(* PLC project paper-machine, Generated TextualNotationConverter 1.0 *)
(* stored: creationDateTime 2025-07-30T12:00:00, modificationDateTime 2025-01-30T12:00:00 *)

FUNCTION_BLOCK ANALOG_IN
  VAR_INPUT
    Name : STRING;
    Description : STRING;
    Raw_Signal : REAL;
    PV_High : REAL;
    PV_Low : REAL;
    Scaling_Slope : REAL;
    Scaling_Offset : REAL;
    Alarm_Enable : BOOL;
  END_VAR
  VAR_OUTPUT
    PV : REAL;
    High_Alarm : BOOL;
    Low_Alarm : BOOL;
    General_Fault : BOOL;
  END_VAR

            
          
END_FUNCTION_BLOCK

FUNCTION_BLOCK BOOL_IN
  VAR_INPUT
    Name : STRING;
    Description : STRING;
    Bool_In : BOOL;
    Alarm_OnTrue : BOOL;
    Alarm_OnFalse : BOOL;
    Latch_Enable : BOOL;
    Reset_Latch : BOOL;
  END_VAR
  VAR_OUTPUT
    Bool_Out : BOOL;
    Alarm_Active : BOOL;
    Latched_Status : BOOL;
  END_VAR

            
          
END_FUNCTION_BLOCK

FUNCTION_BLOCK MOTOR_VSD
  VAR_INPUT
    Name : STRING;
    Description : STRING;
    Start_Cmd : BOOL;
    Stop_Cmd : BOOL;
    Speed_SP : REAL;
    Accel_Ramp : STRING;
    Decel_Ramp : STRING;
    Inhibit : BOOL;
  END_VAR
  VAR_OUTPUT
    Speed_Out : REAL;
    FB_Running : BOOL;
    FB_Fault : BOOL;
    FB_Ready : BOOL;
    FB_ActualSpeed : REAL;
    Alarm_Speed_Deviation : BOOL;
    Alarm_Comm_Fail : BOOL;
  END_VAR

            
          
END_FUNCTION_BLOCK

FUNCTION_BLOCK PID_BASIC
  VAR_INPUT
    Name : STRING;
    Description : STRING;
    AUTO : BOOL;
    PV : REAL;
    SP : REAL;
    MV_MIN : REAL;
    MV_MAX : REAL;
    X0 : REAL;
    KP : REAL;
    TR : REAL;
    TD : REAL;
    PV_High : REAL;
    PV_Low : REAL;
    Deviation_Limit : REAL;
    Inhibit : BOOL;
  END_VAR
  VAR_OUTPUT
    PV_High_Alarm : BOOL;
    PV_Low_Alarm : BOOL;
    Deviation_Alarm : BOOL;
    XOUT : REAL;
  END_VAR

            
          
END_FUNCTION_BLOCK

FUNCTION_BLOCK VALVE_ELECTRIC
  VAR_INPUT
    Name : STRING;
    Description : STRING;
    Control_Signal : REAL;
    Manual_Mode : BOOL;
    Manual_Position : REAL;
    Open_Limit : REAL;
    Close_Limit : REAL;
    Timeout : STRING;
    Inhibit : BOOL;
  END_VAR
  VAR_OUTPUT
    Valve_Position : REAL;
    Feedback_Pos : REAL;
    Valve_Moving : BOOL;
    Position_Error : BOOL;
    Alarm : BOOL;
  END_VAR

            
          
END_FUNCTION_BLOCK

FUNCTION_BLOCK VALVE_ON_OFF
  VAR_INPUT
    Name : STRING;
    Description : STRING;
    Open_Cmd : BOOL;
    Close_Cmd : BOOL;
    Timeout : STRING;
    Inhibit : BOOL;
  END_VAR
  VAR_OUTPUT
    FB_Opened : BOOL;
    FB_Closed : BOOL;
    Valve_Open_Out : BOOL;
    Valve_Close_Out : BOOL;
    Alarm_Position_Error : BOOL;
    Alarm_General : BOOL;
  END_VAR

            
          
END_FUNCTION_BLOCK

PROGRAM Section2
  VAR
    LT101_Flow_PV_m3ph : REAL;
    FC101_MV_Percent : REAL;
    HopperLevel_Above20 : BOOL;
  END_VAR
  VAR
    LT-101 : ANALOG_IN;
    FC-101 : PID_BASIC;
    M-102 : MOTOR_VSD;
    FV-106 : VALVE_ELECTRIC;
    XV-102 : VALVE_ON_OFF;
    XV-104 : VALVE_ON_OFF;
    XV-105 : VALVE_ON_OFF;
    ILK-FC-101-XV-102-OPEN : BOOL_IN;
    ILK-FC-101-XV-104-OPEN : BOOL_IN;
    ILK-FC-101-LT-101-VALID : BOOL_IN;
    PERM-M-102-LEVEL-ABOVE-20 : BOOL_IN;
    PERM-M-102-XV-105-CLOSED : BOOL_IN;
    M102RestartDelay_TON : TON;
  END_VAR
  VAR  (* added by the conversion: wires and edge detectors of the diagram *)
    _OR9_OUT : BOOL;
    _NOT10_OUT : BOOL;
    _AND3_OUT : BOOL;
  END_VAR

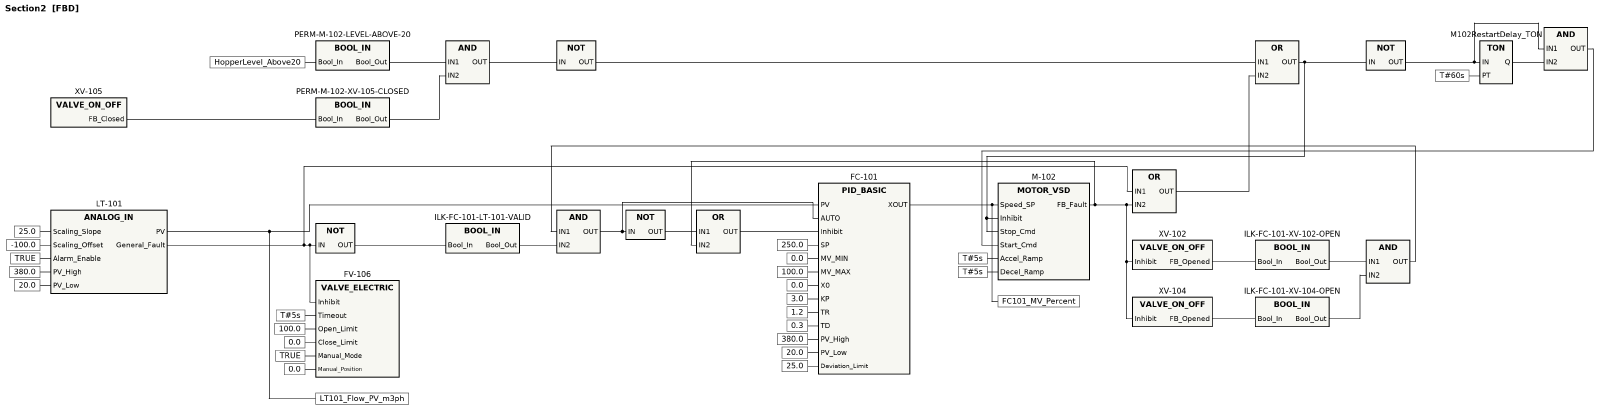
(* FBD diagram, written out as Structured Text *)
LT-101(Scaling_Slope := 25.0, Scaling_Offset := -100.0, Alarm_Enable := TRUE, PV_High := 380.0, PV_Low := 20.0);
PERM-M-102-LEVEL-ABOVE-20(Bool_In := HopperLevel_Above20);
XV-105();
PERM-M-102-XV-105-CLOSED(Bool_In := XV-105.FB_Closed);
_OR9_OUT := NOT (PERM-M-102-LEVEL-ABOVE-20.Bool_Out AND PERM-M-102-XV-105-CLOSED.Bool_Out) OR LT-101.General_Fault OR M-102.FB_Fault;
_NOT10_OUT := NOT _OR9_OUT;
M102RestartDelay_TON(IN := _NOT10_OUT, PT := T#60s);
M-102(Speed_SP := FC-101.XOUT, Inhibit := _OR9_OUT, Stop_Cmd := _OR9_OUT, Start_Cmd := _NOT10_OUT AND M102RestartDelay_TON.Q, Accel_Ramp := T#5s, Decel_Ramp := T#5s);
XV-102(Inhibit := M-102.FB_Fault);
ILK-FC-101-XV-102-OPEN(Bool_In := XV-102.FB_Opened);
XV-104(Inhibit := M-102.FB_Fault);
ILK-FC-101-XV-104-OPEN(Bool_In := XV-104.FB_Opened);
ILK-FC-101-LT-101-VALID(Bool_In := NOT LT-101.General_Fault);
_AND3_OUT := ILK-FC-101-XV-102-OPEN.Bool_Out AND ILK-FC-101-XV-104-OPEN.Bool_Out AND ILK-FC-101-LT-101-VALID.Bool_Out;
FC-101(PV := LT-101.PV, AUTO := _AND3_OUT, Inhibit := NOT _AND3_OUT OR M-102.FB_Fault, SP := 250.0, MV_MIN := 0.0, MV_MAX := 100.0, X0 := 0.0, KP := 3.0, TR := 1.2, TD := 0.3, PV_High := 380.0, PV_Low := 20.0, Deviation_Limit := 25.0);
FC101_MV_Percent := FC-101.XOUT;
LT101_Flow_PV_m3ph := LT-101.PV;
FV-106(Inhibit := LT-101.General_Fault, Timeout := T#5s, Open_Limit := 100.0, Close_Limit := 0.0, Manual_Mode := TRUE, Manual_Position := 0.0);
END_PROGRAM

FUNCTION_BLOCK DIGITAL_IN
  VAR_INPUT
    Name : STRING;
    Description : STRING;
    DI_Raw : BOOL;
    DebounceTime : STRING;
    EnableAlarm : BOOL;
  END_VAR
  VAR_OUTPUT
    DI_Out : BOOL;
    Fault_State : BOOL;
  END_VAR

            
          
END_FUNCTION_BLOCK

FUNCTION_BLOCK DUTY_STANDBY
  VAR_INPUT
    Name : STRING;
    Description : STRING;
    Enable : BOOL;
    StartRequest : BOOL;
    AlternateEnable : BOOL;
    ForcePumpA : BOOL;
    ForcePumpB : BOOL;
    DutyElapsed : BOOL;
    MinRunElapsed : BOOL;
    SwitchoverDelayElapsed : BOOL;
    StartTimeoutElapsed : BOOL;
    PumpA_RunFB : BOOL;
    PumpB_RunFB : BOOL;
    PumpA_Fault : BOOL;
    PumpB_Fault : BOOL;
    Reset : BOOL;
    Inhibit : BOOL;
  END_VAR
  VAR_OUTPUT
    CmdPumpA : BOOL;
    CmdPumpB : BOOL;
    ActiveIsA : BOOL;
    SwitchedDueToDuty : BOOL;
    SwitchedDueToFailure : BOOL;
    Alarm_FailedStart_A : BOOL;
    Alarm_FailedStart_B : BOOL;
    Alarm_NoAvailablePump : BOOL;
  END_VAR

            
          
END_FUNCTION_BLOCK

FUNCTION_BLOCK MOTOR_2SPD
  VAR_INPUT
    Name : STRING;
    Description : STRING;
    Start_Cmd : BOOL;
    Stop_Cmd : BOOL;
    Speed_High_Cmd : BOOL;
    Speed_Low_Cmd : BOOL;
    Inhibit : BOOL;
  END_VAR
  VAR_OUTPUT
    Motor_Start_Out : BOOL;
    FB_Running : BOOL;
    FB_Trip : BOOL;
    FB_HighSpeed : BOOL;
    FB_LowSpeed : BOOL;
    Alarm_Speed_Error : BOOL;
  END_VAR

            
          
END_FUNCTION_BLOCK

FUNCTION_BLOCK MOTOR_ON_OFF
  VAR_INPUT
    Name : STRING;
    Description : STRING;
    Start_Cmd : BOOL;
    Stop_Cmd : BOOL;
    Start_Delay : STRING;
    MinRunTime : STRING;
    Inhibit : BOOL;
  END_VAR
  VAR_OUTPUT
    Motor_Start_Out : BOOL;
    FB_Running : BOOL;
    FB_Trip : BOOL;
    Alarm_Start_Fail : BOOL;
    Alarm_Stop_Fail : BOOL;
  END_VAR

            
          
END_FUNCTION_BLOCK

FUNCTION_BLOCK RATIO_CONTROL
  VAR_INPUT
    Name : STRING;
    Description : STRING;
    Auto : BOOL;
    PrimaryPV : REAL;
    SecondaryPV : REAL;
    RatioSP : REAL;
    Bias : REAL;
    TrimKp : REAL;
    TrimTi : STRING;
    MV_MIN : REAL;
    MV_MAX : REAL;
    ManOut : REAL;
    Inhibit : BOOL;
  END_VAR
  VAR_OUTPUT
    SlaveSP : REAL;
    ActiveRatio : REAL;
    RatioErr : REAL;
  END_VAR

            
          
END_FUNCTION_BLOCK

FUNCTION_BLOCK SPLIT_RANGE
  VAR_INPUT
    Name : STRING;
    Description : STRING;
    IN : REAL;
    Split_Point : REAL;
    Output1_Start : REAL;
    Output1_End : REAL;
    Output2_Start : REAL;
    Output2_End : REAL;
  END_VAR
  VAR_OUTPUT
    OUT1 : REAL;
    OUT2 : REAL;
  END_VAR

            
          
END_FUNCTION_BLOCK

FUNCTION_BLOCK VOTING_ANALOG
  VAR_INPUT
    Name : STRING;
    Description : STRING;
    Input1 : REAL;
    Input2 : REAL;
    Input3 : REAL;
    Deviation_Limit : REAL;
    Voting_Scheme : STRING;
    EnableAlarm : BOOL;
    Inhibit : BOOL;
  END_VAR
  VAR_OUTPUT
    Voted_Output : REAL;
    Sensor1_Fault : BOOL;
    Sensor2_Fault : BOOL;
    Sensor3_Fault : BOOL;
    Alarm_Voting_Error : BOOL;
    Healthy_Sensors_Count : INT;
  END_VAR

            
          
END_FUNCTION_BLOCK

PROGRAM Section3
  VAR
    TIC104_RSP_to_FC203 : REAL;
    PIC101_RSP_to_FC202 : REAL;
    FC203_ControlSignal_SV203 : REAL;
    FC202_ControlSignal_FV202 : REAL;
  END_VAR
  VAR
    PT-101 : ANALOG_IN;
    TT-103 : ANALOG_IN;
    PIC-101 : PID_BASIC;
    TIC-104 : PID_BASIC;
    FC-202 : PID_BASIC;
    FC-203 : PID_BASIC;
    FV-202 : VALVE_ELECTRIC;
    SV-203 : VALVE_ELECTRIC;
  END_VAR
  VAR  (* added by the conversion: wires and edge detectors of the diagram *)
    _OR51_OUT : BOOL;
  END_VAR

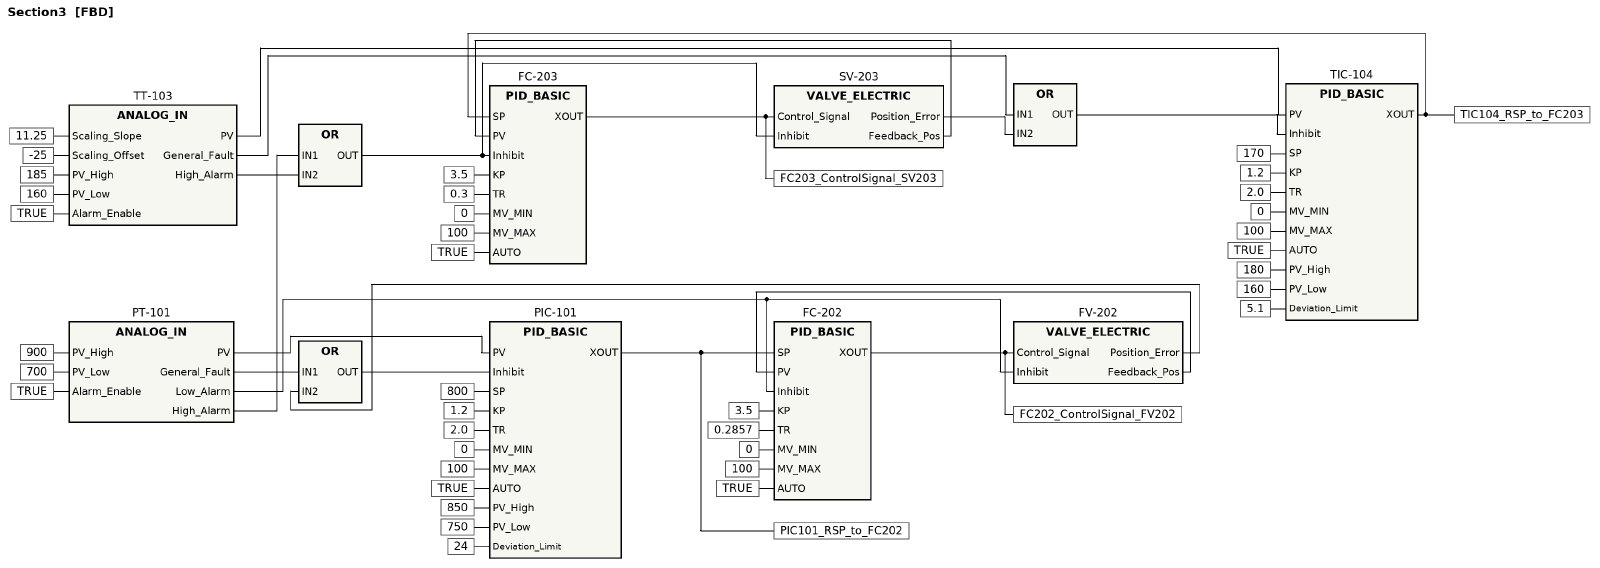
(* FBD diagram, written out as Structured Text *)
PT-101(PV_High := 900, PV_Low := 700, Alarm_Enable := TRUE);
FV-202(Control_Signal := FC-202.XOUT, Inhibit := PT-101.Low_Alarm);
PIC-101(PV := PT-101.PV, Inhibit := PT-101.General_Fault OR FV-202.Position_Error, SP := 800, KP := 1.2, TR := 2.0, MV_MIN := 0, MV_MAX := 100, AUTO := TRUE, PV_High := 850, PV_Low := 750, Deviation_Limit := 24);
FC-202(SP := PIC-101.XOUT, PV := FV-202.Feedback_Pos, Inhibit := PT-101.Low_Alarm, KP := 3.5, TR := 0.2857, MV_MIN := 0, MV_MAX := 100, AUTO := TRUE);
FC202_ControlSignal_FV202 := FC-202.XOUT;
TT-103(Scaling_Slope := 11.25, Scaling_Offset := -25, PV_High := 185, PV_Low := 160, Alarm_Enable := TRUE);
_OR51_OUT := PT-101.High_Alarm OR TT-103.High_Alarm;
SV-203(Control_Signal := FC-203.XOUT, Inhibit := _OR51_OUT);
TIC-104(PV := TT-103.PV, Inhibit := TT-103.General_Fault OR SV-203.Position_Error, SP := 170, KP := 1.2, TR := 2.0, MV_MIN := 0, MV_MAX := 100, AUTO := TRUE, PV_High := 180, PV_Low := 160, Deviation_Limit := 5.1);
FC-203(SP := TIC-104.XOUT, PV := SV-203.Feedback_Pos, Inhibit := _OR51_OUT, KP := 3.5, TR := 0.3, MV_MIN := 0, MV_MAX := 100, AUTO := TRUE);
FC203_ControlSignal_SV203 := FC-203.XOUT;
PIC101_RSP_to_FC202 := PIC-101.XOUT;
TIC104_RSP_to_FC203 := TIC-104.XOUT;
END_PROGRAM

PROGRAM Section4
  VAR
    PIT103_Pressure_PV : REAL;
    PT101_UpstreamPressure_PV : REAL;
    DT301_Density_PV : REAL;
    PIC104_MV_to_FV106 : REAL;
    FV106_Position_Feedback : REAL;
  END_VAR
  VAR
    PIT-103 : ANALOG_IN;
    PT-101 : ANALOG_IN;
    DT-301 : ANALOG_IN;
    PIC-104 : PID_BASIC;
    FV-106 : VALVE_ELECTRIC;
    XV-102 : VALVE_ON_OFF;
    XV-107 : VALVE_ON_OFF;
    XV-102-OPEN-LS : DIGITAL_IN;
    XV-107-OPEN-LS : DIGITAL_IN;
    ILK-FEED-PRESSURE-OK : BOOL_IN;
    ILK-OVERPRESSURE-TRIP : BOOL_IN;
    ILK-DENSITY-OK : BOOL_IN;
    ILK-XV102-OPEN : BOOL_IN;
    ILK-XV107-OPEN : BOOL_IN;
    ILK-SYSTEM-FAULT : BOOL_IN;
  END_VAR

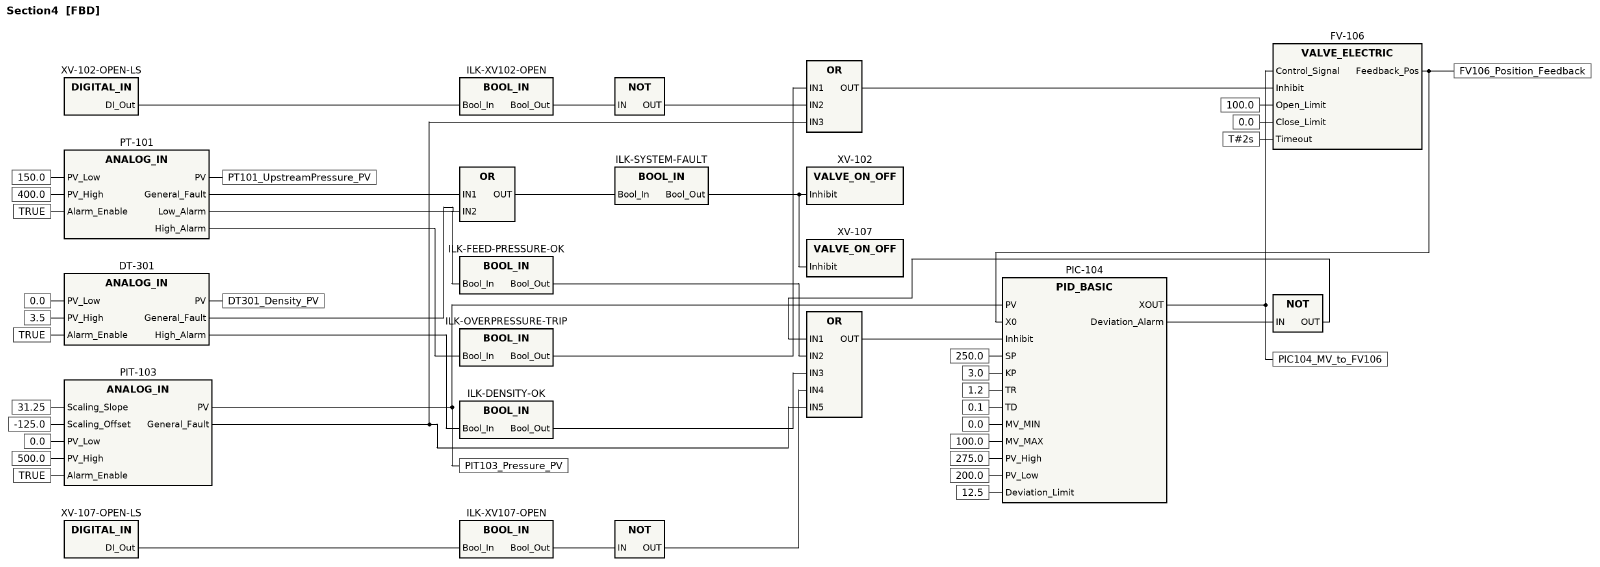
(* FBD diagram, written out as Structured Text *)
DT-301(PV_Low := 0.0, PV_High := 3.5, Alarm_Enable := TRUE);
DT301_Density_PV := DT-301.PV;
PIT-103(Scaling_Slope := 31.25, Scaling_Offset := -125.0, PV_Low := 0.0, PV_High := 500.0, Alarm_Enable := TRUE);
PT-101(PV_Low := 150.0, PV_High := 400.0, Alarm_Enable := TRUE);
ILK-FEED-PRESSURE-OK(Bool_In := PT-101.Low_Alarm);
ILK-DENSITY-OK(Bool_In := DT-301.High_Alarm);
XV-107-OPEN-LS();
ILK-XV107-OPEN(Bool_In := XV-107-OPEN-LS.DI_Out);
PIC-104(PV := PIT-103.PV, X0 := FV-106.Feedback_Pos, Inhibit := NOT PIC-104.Deviation_Alarm OR ILK-FEED-PRESSURE-OK.Bool_Out OR ILK-DENSITY-OK.Bool_Out OR NOT ILK-XV107-OPEN.Bool_Out OR PIT-103.General_Fault, SP := 250.0, KP := 3.0, TR := 1.2, TD := 0.1, MV_MIN := 0.0, MV_MAX := 100.0, PV_High := 275.0, PV_Low := 200.0, Deviation_Limit := 12.5);
ILK-OVERPRESSURE-TRIP(Bool_In := PT-101.High_Alarm);
XV-102-OPEN-LS();
ILK-XV102-OPEN(Bool_In := XV-102-OPEN-LS.DI_Out);
FV-106(Control_Signal := PIC-104.XOUT, Inhibit := ILK-OVERPRESSURE-TRIP.Bool_Out OR NOT ILK-XV102-OPEN.Bool_Out OR PIT-103.General_Fault, Open_Limit := 100.0, Close_Limit := 0.0, Timeout := T#2s);
FV106_Position_Feedback := FV-106.Feedback_Pos;
PIC104_MV_to_FV106 := PIC-104.XOUT;
PIT103_Pressure_PV := PIT-103.PV;
PT101_UpstreamPressure_PV := PT-101.PV;
ILK-SYSTEM-FAULT(Bool_In := PT-101.General_Fault OR DT-301.General_Fault);
XV-102(Inhibit := ILK-SYSTEM-FAULT.Bool_Out);
XV-107(Inhibit := ILK-SYSTEM-FAULT.Bool_Out);
END_PROGRAM

PROGRAM Section5
  VAR
    AT102_pH_PV : REAL;
    AT107_pH_PV : REAL;
    TIT106_Temperature_PV : REAL;
    FIT_UPSTREAM_Flow_PV : REAL;
    DPIT_FLOW_PV : REAL;
    PIT_DOWNSTREAM_Pressure_PV : REAL;
    LIT_TOWER_Level_PV : REAL;
    LIC102_MV_to_FV101 : REAL;
    TIC106_MV_to_FV103 : REAL;
    LIC104_Output_to_XV104 : REAL;
    FV101_Position_AO : REAL;
    FV103_Position_AO : REAL;
  END_VAR
  VAR
    AT-102 : ANALOG_IN;
    AT-107 : ANALOG_IN;
    TIT-106 : ANALOG_IN;
    FIT-UPSTREAM : ANALOG_IN;
    DPIT-FLOW : ANALOG_IN;
    PIT-DOWNSTREAM : ANALOG_IN;
    LIT-TOWER : ANALOG_IN;
    LIC-102 : PID_BASIC;
    TIC-106 : PID_BASIC;
    LIC-104 : PID_BASIC;
    FV-101 : VALVE_ELECTRIC;
    FV-103 : VALVE_ELECTRIC;
    XV-104 : VALVE_ON_OFF;
    INTERLOCK-FV101-UPSTREAM-FLOW-OK : BOOL_IN;
    INTERLOCK-LIC102-PH-SAFE : BOOL_IN;
    INTERLOCK-TIC106-TEMP-SAFE : BOOL_IN;
    INTERLOCK-LIC104-FLOW-OK : BOOL_IN;
    INTERLOCK-LIC104-PRESSURE-OK : BOOL_IN;
    PERMISSIVE-TOWER-LEVEL-OK : BOOL_IN;
  END_VAR

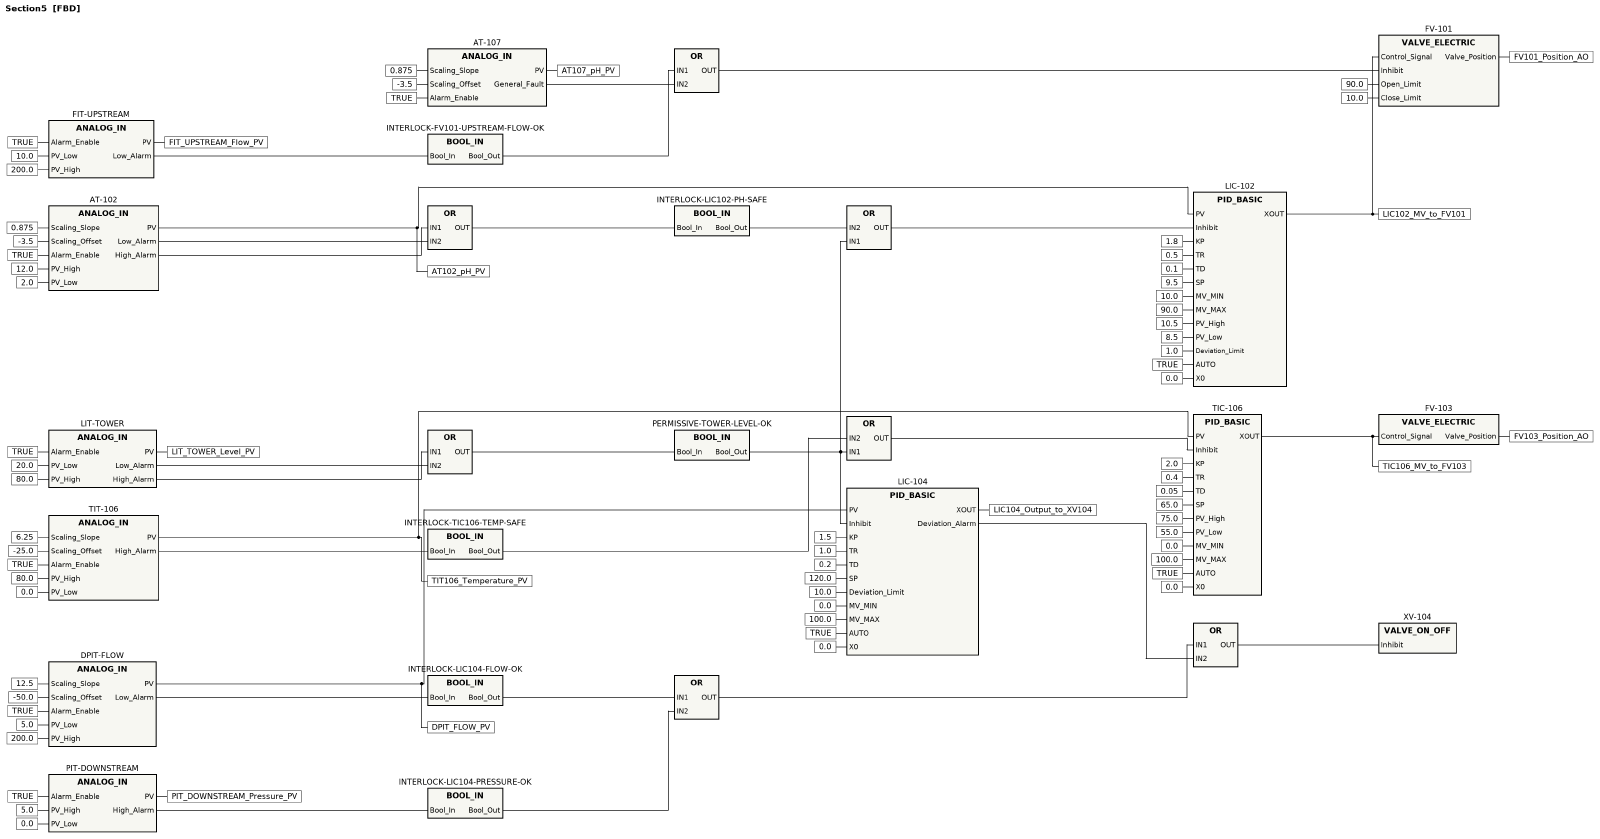
(* FBD diagram, written out as Structured Text *)
AT-102(Scaling_Slope := 0.875, Scaling_Offset := -3.5, Alarm_Enable := TRUE, PV_High := 12.0, PV_Low := 2.0);
AT102_pH_PV := AT-102.PV;
AT-107(Scaling_Slope := 0.875, Scaling_Offset := -3.5, Alarm_Enable := TRUE);
AT107_pH_PV := AT-107.PV;
DPIT-FLOW(Scaling_Slope := 12.5, Scaling_Offset := -50.0, Alarm_Enable := TRUE, PV_Low := 5.0, PV_High := 200.0);
DPIT_FLOW_PV := DPIT-FLOW.PV;
FIT-UPSTREAM(Alarm_Enable := TRUE, PV_Low := 10.0, PV_High := 200.0);
FIT_UPSTREAM_Flow_PV := FIT-UPSTREAM.PV;
INTERLOCK-LIC102-PH-SAFE(Bool_In := AT-102.High_Alarm OR AT-102.Low_Alarm);
LIT-TOWER(Alarm_Enable := TRUE, PV_Low := 20.0, PV_High := 80.0);
PERMISSIVE-TOWER-LEVEL-OK(Bool_In := LIT-TOWER.High_Alarm OR LIT-TOWER.Low_Alarm);
LIC-102(PV := AT-102.PV, Inhibit := INTERLOCK-LIC102-PH-SAFE.Bool_Out OR PERMISSIVE-TOWER-LEVEL-OK.Bool_Out, KP := 1.8, TR := 0.5, TD := 0.1, SP := 9.5, MV_MIN := 10.0, MV_MAX := 90.0, PV_High := 10.5, PV_Low := 8.5, Deviation_Limit := 1.0, AUTO := TRUE, X0 := 0.0);
INTERLOCK-FV101-UPSTREAM-FLOW-OK(Bool_In := FIT-UPSTREAM.Low_Alarm);
FV-101(Control_Signal := LIC-102.XOUT, Inhibit := INTERLOCK-FV101-UPSTREAM-FLOW-OK.Bool_Out OR AT-107.General_Fault, Open_Limit := 90.0, Close_Limit := 10.0);
FV101_Position_AO := FV-101.Valve_Position;
TIT-106(Scaling_Slope := 6.25, Scaling_Offset := -25.0, Alarm_Enable := TRUE, PV_High := 80.0, PV_Low := 0.0);
INTERLOCK-TIC106-TEMP-SAFE(Bool_In := TIT-106.High_Alarm);
TIC-106(PV := TIT-106.PV, Inhibit := INTERLOCK-TIC106-TEMP-SAFE.Bool_Out OR PERMISSIVE-TOWER-LEVEL-OK.Bool_Out, KP := 2.0, TR := 0.4, TD := 0.05, SP := 65.0, PV_High := 75.0, PV_Low := 55.0, MV_MIN := 0.0, MV_MAX := 100.0, AUTO := TRUE, X0 := 0.0);
FV-103(Control_Signal := TIC-106.XOUT);
FV103_Position_AO := FV-103.Valve_Position;
LIC102_MV_to_FV101 := LIC-102.XOUT;
LIC-104(PV := DPIT-FLOW.PV, Inhibit := PERMISSIVE-TOWER-LEVEL-OK.Bool_Out, KP := 1.5, TR := 1.0, TD := 0.2, SP := 120.0, Deviation_Limit := 10.0, MV_MIN := 0.0, MV_MAX := 100.0, AUTO := TRUE, X0 := 0.0);
LIC104_Output_to_XV104 := LIC-104.XOUT;
LIT_TOWER_Level_PV := LIT-TOWER.PV;
PIT-DOWNSTREAM(Alarm_Enable := TRUE, PV_High := 5.0, PV_Low := 0.0);
PIT_DOWNSTREAM_Pressure_PV := PIT-DOWNSTREAM.PV;
TIC106_MV_to_FV103 := TIC-106.XOUT;
TIT106_Temperature_PV := TIT-106.PV;
INTERLOCK-LIC104-FLOW-OK(Bool_In := DPIT-FLOW.Low_Alarm);
INTERLOCK-LIC104-PRESSURE-OK(Bool_In := PIT-DOWNSTREAM.High_Alarm);
XV-104(Inhibit := INTERLOCK-LIC104-FLOW-OK.Bool_Out OR INTERLOCK-LIC104-PRESSURE-OK.Bool_Out OR LIC-104.Deviation_Alarm);
END_PROGRAM

PROGRAM Section6
  VAR
    SELC_501_MV_Percent : REAL;
    FC_502_MV_Percent : REAL;
  END_VAR
  VAR
    CT-501 : ANALOG_IN;
    LT-501 : ANALOG_IN;
    PT-502 : ANALOG_IN;
    PG-501 : ANALOG_IN;
    SEL-501 : ANALOG_IN;
    FC-502 : PID_BASIC;
    SELC-501 : PID_BASIC;
    FV-502 : VALVE_ELECTRIC;
    PGA-501 : VALVE_ELECTRIC;
    M-501 : MOTOR_ON_OFF;
  END_VAR
  VAR  (* added by the conversion: wires and edge detectors of the diagram *)
    _OR250_OUT : BOOL;
    _OR248_OUT : BOOL;
    _OR253_OUT : BOOL;
  END_VAR

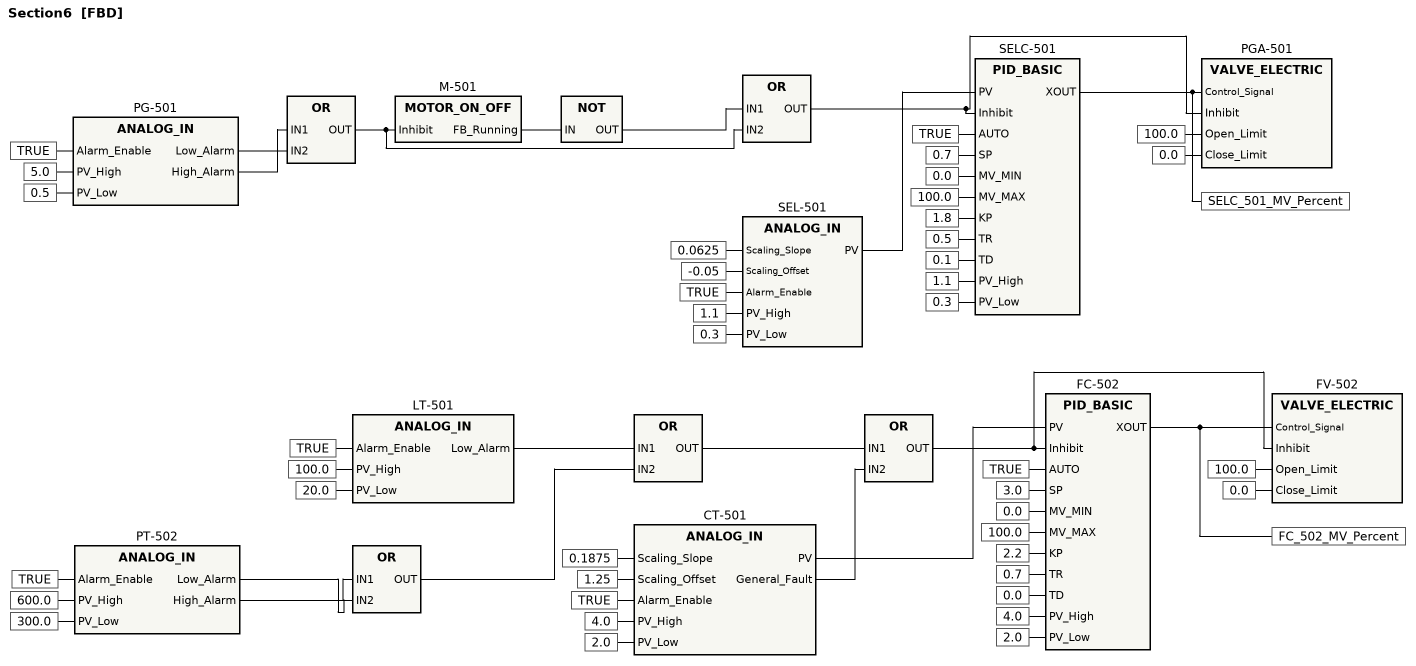
(* FBD diagram, written out as Structured Text *)
CT-501(Scaling_Slope := 0.1875, Scaling_Offset := 1.25, Alarm_Enable := TRUE, PV_High := 4.0, PV_Low := 2.0);
LT-501(Alarm_Enable := TRUE, PV_High := 100.0, PV_Low := 20.0);
PT-502(Alarm_Enable := TRUE, PV_High := 600.0, PV_Low := 300.0);
_OR250_OUT := LT-501.Low_Alarm OR PT-502.High_Alarm OR PT-502.Low_Alarm OR CT-501.General_Fault;
FC-502(PV := CT-501.PV, Inhibit := _OR250_OUT, AUTO := TRUE, SP := 3.0, MV_MIN := 0.0, MV_MAX := 100.0, KP := 2.2, TR := 0.7, TD := 0.0, PV_High := 4.0, PV_Low := 2.0);
FC_502_MV_Percent := FC-502.XOUT;
SEL-501(Scaling_Slope := 0.0625, Scaling_Offset := -0.05, Alarm_Enable := TRUE, PV_High := 1.1, PV_Low := 0.3);
PG-501(Alarm_Enable := TRUE, PV_High := 5.0, PV_Low := 0.5);
_OR248_OUT := PG-501.High_Alarm OR PG-501.Low_Alarm;
M-501(Inhibit := _OR248_OUT);
_OR253_OUT := NOT M-501.FB_Running OR _OR248_OUT;
SELC-501(PV := SEL-501.PV, Inhibit := _OR253_OUT, AUTO := TRUE, SP := 0.7, MV_MIN := 0.0, MV_MAX := 100.0, KP := 1.8, TR := 0.5, TD := 0.1, PV_High := 1.1, PV_Low := 0.3);
SELC_501_MV_Percent := SELC-501.XOUT;
FV-502(Control_Signal := FC-502.XOUT, Inhibit := _OR250_OUT, Open_Limit := 100.0, Close_Limit := 0.0);
PGA-501(Control_Signal := SELC-501.XOUT, Inhibit := _OR253_OUT, Open_Limit := 100.0, Close_Limit := 0.0);
END_PROGRAM

PROGRAM Section7
  VAR
    FT601_Flow_SP : REAL;
    Ratio_Bias : REAL;
  END_VAR
  VAR
    CT-601 : ANALOG_IN;
    FT-601 : ANALOG_IN;
    PIT-601 : ANALOG_IN;
    VT-601 : ANALOG_IN;
    FIC-601 : PID_BASIC;
    FFIC-601 : RATIO_CONTROL;
    FV-601 : VALVE_ELECTRIC;
    P-601 : MOTOR_ON_OFF;
    FS-601 : BOOL_IN;
    P-601-RUN : BOOL_IN;
    PIT-601-OK : BOOL_IN;
    VT-601-OK : BOOL_IN;
    ALM-601 : DIGITAL_IN;
    ALM-602 : DIGITAL_IN;
    ALM-603 : DIGITAL_IN;
    ALM-604 : DIGITAL_IN;
  END_VAR
  VAR  (* added by the conversion: wires and edge detectors of the diagram *)
    _NOT310_OUT : BOOL;
    _OR311_OUT : BOOL;
    _NOT314_OUT : BOOL;
    _OR312_OUT : BOOL;
  END_VAR

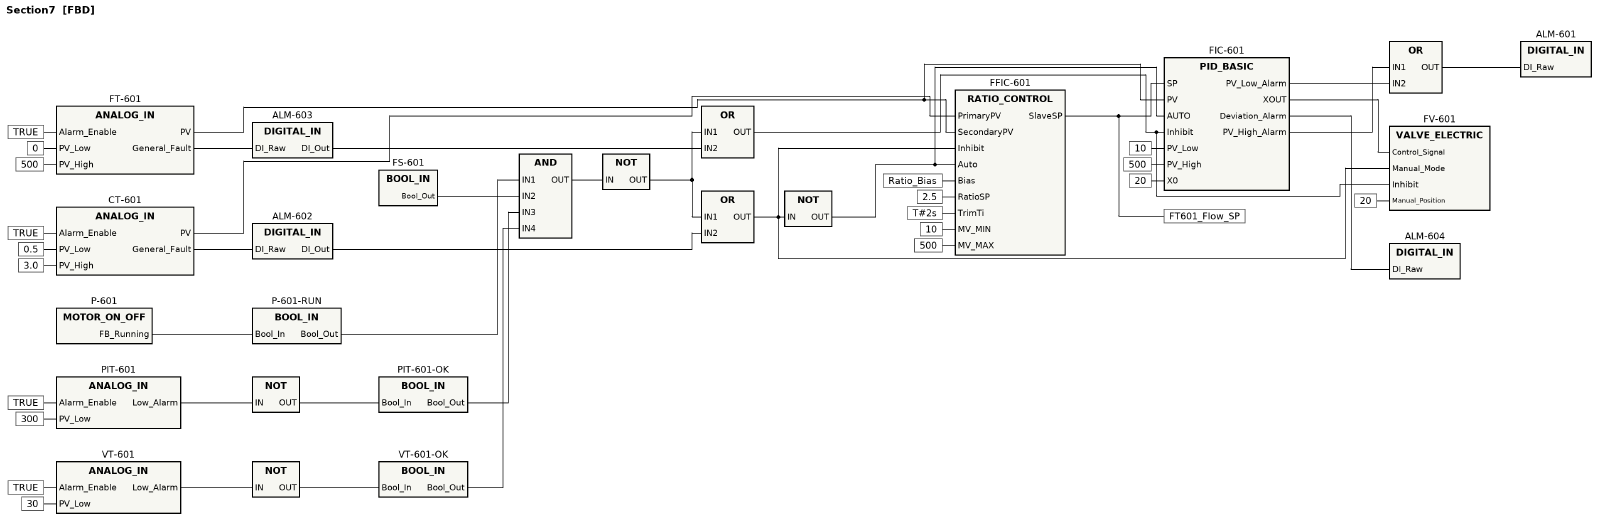
(* FBD diagram, written out as Structured Text *)
CT-601(Alarm_Enable := TRUE, PV_Low := 0.5, PV_High := 3.0);
FT-601(Alarm_Enable := TRUE, PV_Low := 0, PV_High := 500);
P-601();
P-601-RUN(Bool_In := P-601.FB_Running);
FS-601();
PIT-601(Alarm_Enable := TRUE, PV_Low := 300);
PIT-601-OK(Bool_In := NOT PIT-601.Low_Alarm);
VT-601(Alarm_Enable := TRUE, PV_Low := 30);
VT-601-OK(Bool_In := NOT VT-601.Low_Alarm);
_NOT310_OUT := NOT (P-601-RUN.Bool_Out AND FS-601.Bool_Out AND PIT-601-OK.Bool_Out AND VT-601-OK.Bool_Out);
ALM-602(DI_Raw := CT-601.General_Fault);
_OR311_OUT := _NOT310_OUT OR ALM-602.DI_Out;
_NOT314_OUT := NOT _OR311_OUT;
FFIC-601(PrimaryPV := CT-601.PV, SecondaryPV := FT-601.PV, Inhibit := _OR311_OUT, Auto := _NOT314_OUT, Bias := Ratio_Bias, RatioSP := 2.5, TrimTi := T#2s, MV_MIN := 10, MV_MAX := 500);
FT601_Flow_SP := FFIC-601.SlaveSP;
ALM-603(DI_Raw := FT-601.General_Fault);
_OR312_OUT := _NOT310_OUT OR ALM-603.DI_Out;
FIC-601(SP := FFIC-601.SlaveSP, PV := FT-601.PV, AUTO := _NOT314_OUT, Inhibit := _OR312_OUT, PV_Low := 10, PV_High := 500, X0 := 20);
FV-601(Control_Signal := FIC-601.XOUT, Manual_Mode := _OR311_OUT, Inhibit := _OR312_OUT, Manual_Position := 20);
ALM-601(DI_Raw := FIC-601.PV_High_Alarm OR FIC-601.PV_Low_Alarm);
ALM-604(DI_Raw := FIC-601.Deviation_Alarm);
END_PROGRAM

PROGRAM Section8
  VAR
    MM701_SheetMoisture_PV : REAL;
    PT701_HydraulicPressure_PV : REAL;
    TT102_PressSectionTemperature_PV : REAL;
    LIC701_ControlOutput_MV_Percent : REAL;
    PV101_ValvePosition_Feedback_Percent : REAL;
    CS701_ControlSwitch_State : BOOL;
    HS701_ManualOverride_State : BOOL;
    SB701_SheetBreak_Status : BOOL;
  END_VAR
  VAR
    MM-701 : ANALOG_IN;
    PT-701 : ANALOG_IN;
    TT-102 : ANALOG_IN;
    CS-701 : BOOL_IN;
    HS-701 : BOOL_IN;
    SB-701 : BOOL_IN;
    LIC-701 : PID_BASIC;
    PV-101 : VALVE_ELECTRIC;
  END_VAR
  VAR  (* added by the conversion: wires and edge detectors of the diagram *)
    _OR353_OUT : BOOL;
  END_VAR

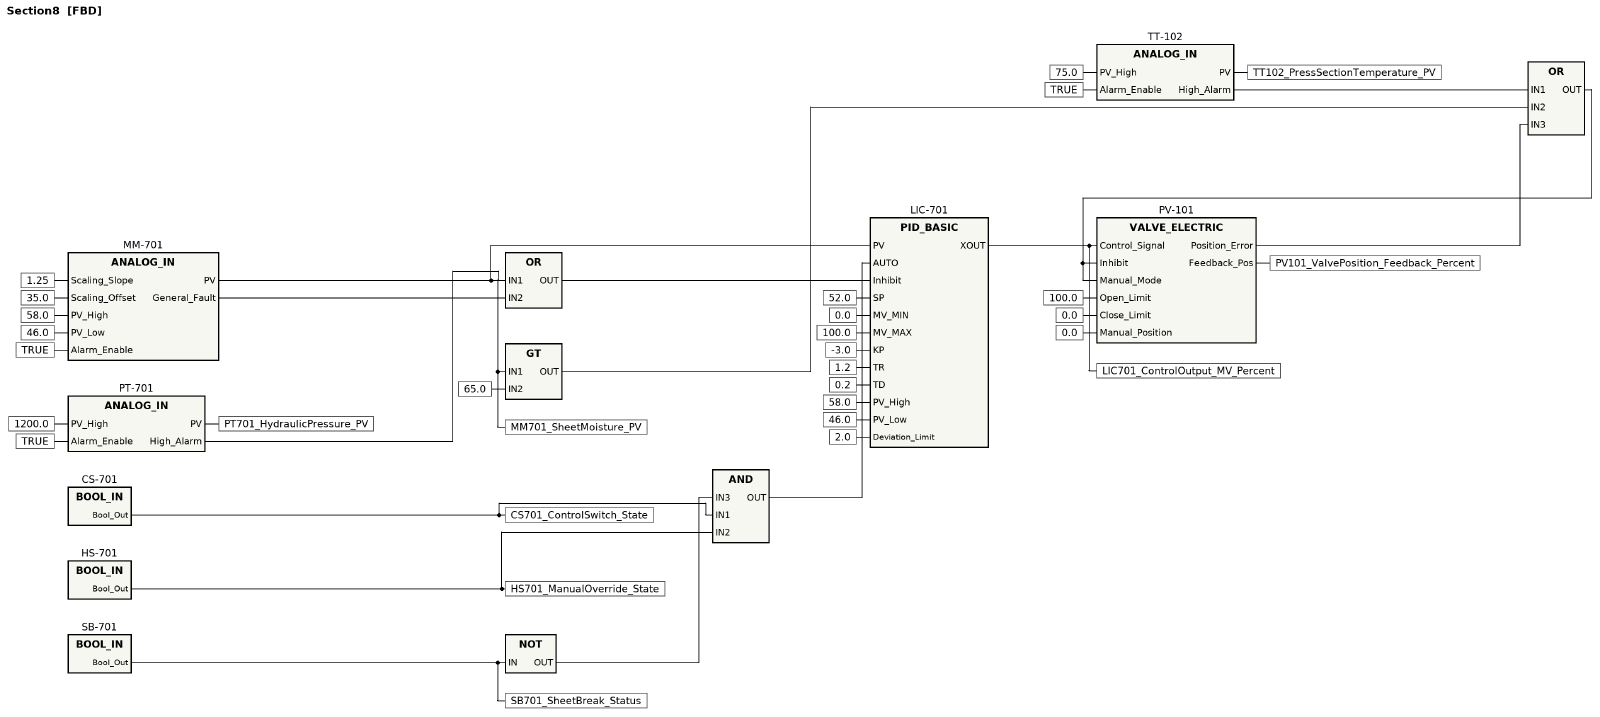
(* FBD diagram, written out as Structured Text *)
CS-701();
CS701_ControlSwitch_State := CS-701.Bool_Out;
HS-701();
HS701_ManualOverride_State := HS-701.Bool_Out;
MM-701(Scaling_Slope := 1.25, Scaling_Offset := 35.0, PV_High := 58.0, PV_Low := 46.0, Alarm_Enable := TRUE);
SB-701();
PT-701(PV_High := 1200.0, Alarm_Enable := TRUE);
LIC-701(PV := MM-701.PV, AUTO := NOT SB-701.Bool_Out AND CS-701.Bool_Out AND HS-701.Bool_Out, Inhibit := PT-701.High_Alarm OR MM-701.General_Fault, SP := 52.0, MV_MIN := 0.0, MV_MAX := 100.0, KP := -3.0, TR := 1.2, TD := 0.2, PV_High := 58.0, PV_Low := 46.0, Deviation_Limit := 2.0);
LIC701_ControlOutput_MV_Percent := LIC-701.XOUT;
MM701_SheetMoisture_PV := MM-701.PV;
PT701_HydraulicPressure_PV := PT-701.PV;
TT-102(PV_High := 75.0, Alarm_Enable := TRUE);
_OR353_OUT := TT-102.High_Alarm OR MM-701.PV > 65.0 OR PV-101.Position_Error;
PV-101(Control_Signal := LIC-701.XOUT, Inhibit := _OR353_OUT, Manual_Mode := _OR353_OUT, Open_Limit := 100.0, Close_Limit := 0.0, Manual_Position := 0.0);
PV101_ValvePosition_Feedback_Percent := PV-101.Feedback_Pos;
SB701_SheetBreak_Status := SB-701.Bool_Out;
TT102_PressSectionTemperature_PV := TT-102.PV;
END_PROGRAM

PROGRAM Section9
  VAR
    F801_VFD_Speed_Cmd_Pct : REAL;
    FV801_SteamFlow_ValvePos_Cmd_Pct : REAL;
    XV802_HoodDamper_Pos_Cmd_Pct : REAL;
    M801_Drive_Torque_Cmd_Pct : REAL;
  END_VAR
  VAR
    TT-801 : ANALOG_IN;
    TT-802 : ANALOG_IN;
    PT-801 : ANALOG_IN;
    IR-801 : ANALOG_IN;
    WT-801 : ANALOG_IN;
    F-801 : MOTOR_VSD;
    M-801 : MOTOR_VSD;
    FV-801 : VALVE_ELECTRIC;
    XV-802 : VALVE_ELECTRIC;
    TC-801 : PID_BASIC;
    SC-801_LOOP : PID_BASIC;
    IR-801_LOOP : PID_BASIC;
    WT-801_LOOP : PID_BASIC;
    PT-801_Overpressure : BOOL_IN;
    IR-801_Available : BOOL_IN;
    XV-802_Open : BOOL_IN;
    TT-802_InRange : BOOL_IN;
    WT-801_InRange : BOOL_IN;
    M-801_Running : BOOL_IN;
  END_VAR
  VAR  (* added by the conversion: wires and edge detectors of the diagram *)
    _OR395_OUT : BOOL;
    _OR394_OUT : BOOL;
    _OR402_OUT : BOOL;
    _NOT400_OUT : BOOL;
  END_VAR

(* FBD diagram, written out as Structured Text *)
IR-801(Scaling_Slope := 0.625, Scaling_Offset := -2.5, PV_High := 5.0, PV_Low := 0, Alarm_Enable := TRUE);
_OR395_OUT := IR-801.General_Fault OR IR-801.Low_Alarm OR IR-801.High_Alarm;
IR-801_LOOP(PV := IR-801.PV, Inhibit := _OR395_OUT, SP := 4.5, KP := 1.8, TR := 0.6, TD := 0.05, MV_MIN := 0, MV_MAX := 100, Deviation_Limit := 0.2, PV_High := 5.0, PV_Low := 0, AUTO := TRUE);
F-801(Speed_SP := IR-801_LOOP.XOUT, Inhibit := _OR395_OUT);
F801_VFD_Speed_Cmd_Pct := F-801.Speed_Out;
TT-801(Scaling_Slope := 9.375, Scaling_Offset := -37.5, PV_High := 125, PV_Low := 0, Alarm_Enable := TRUE);
PT-801(PV_High := 900, PV_Low := 600, Alarm_Enable := TRUE);
PT-801_Overpressure(Bool_In := PT-801.High_Alarm);
_OR394_OUT := PT-801_Overpressure.Bool_Out OR PT-801.Low_Alarm OR TT-801.High_Alarm;
SC-801_LOOP(PV := TT-801.PV, Inhibit := _OR394_OUT, SP := 115, KP := 3.0, TR := 0.5, TD := 0.1, MV_MIN := 0, MV_MAX := 100, PV_High := 125, PV_Low := 0, AUTO := TRUE);
FV-801(Control_Signal := SC-801_LOOP.XOUT, Inhibit := _OR394_OUT, Open_Limit := 100, Close_Limit := 0, Manual_Mode := FALSE);
FV801_SteamFlow_ValvePos_Cmd_Pct := FV-801.Valve_Position;
WT-801(Scaling_Slope := 31.25, Scaling_Offset := -125, PV_High := 450, PV_Low := 50, Alarm_Enable := TRUE);
M-801_Running(Bool_In := M-801.FB_Running);
_OR402_OUT := WT-801.High_Alarm OR WT-801.Low_Alarm;
WT-801_InRange(Bool_In := NOT _OR402_OUT);
WT-801_LOOP(PV := WT-801.PV, Inhibit := NOT (M-801_Running.Bool_Out AND WT-801_InRange.Bool_Out), SP := 250, KP := 4.0, TR := 1.0, TD := 0.3, MV_MIN := 0, MV_MAX := 100, PV_High := 400, PV_Low := 50, AUTO := TRUE);
M-801(Speed_SP := WT-801_LOOP.XOUT, Inhibit := _OR402_OUT);
M801_Drive_Torque_Cmd_Pct := M-801.Speed_Out;
TT-802(Scaling_Slope := 4.375, Scaling_Offset := 32.5, PV_High := 120, PV_Low := 50, Alarm_Enable := TRUE);
XV-802_Open(Bool_In := XV-802.Feedback_Pos > 20);
TT-802_InRange(Bool_In := NOT (TT-802.High_Alarm OR TT-802.Low_Alarm));
_NOT400_OUT := NOT (XV-802_Open.Bool_Out AND TT-802_InRange.Bool_Out);
TC-801(PV := TT-802.PV, Inhibit := _NOT400_OUT, SP := 85, KP := 2.5, TR := 0.8, TD := 0.2, MV_MIN := 10, MV_MAX := 90, PV_High := 95, PV_Low := 50, AUTO := TRUE);
XV-802(Control_Signal := TC-801.XOUT, Inhibit := _NOT400_OUT OR TC-801.PV_High_Alarm, Open_Limit := 90, Close_Limit := 10, Manual_Mode := FALSE);
XV802_HoodDamper_Pos_Cmd_Pct := XV-802.Valve_Position;
IR-801_Available(Bool_In := NOT _OR395_OUT);
END_PROGRAM

PROGRAM Section10
  VAR
    FFIC903_CoatingFlow_SP : REAL;
    FV104_ControlSignal_Pct : REAL;
    FFIC903_RatioSP : REAL;
    FFIC903_RatioBias : REAL;
  END_VAR
  VAR
    FT-901 : ANALOG_IN;
    FT-902 : ANALOG_IN;
    CW-901 : ANALOG_IN;
    FFIC-903 : RATIO_CONTROL;
    FIC-904 : PID_BASIC;
    FV-104 : VALVE_ELECTRIC;
    XV-105 : VALVE_ON_OFF;
  END_VAR
  VAR  (* added by the conversion: wires and edge detectors of the diagram *)
    _OR497_OUT : BOOL;
    _NOT499_OUT : BOOL;
  END_VAR

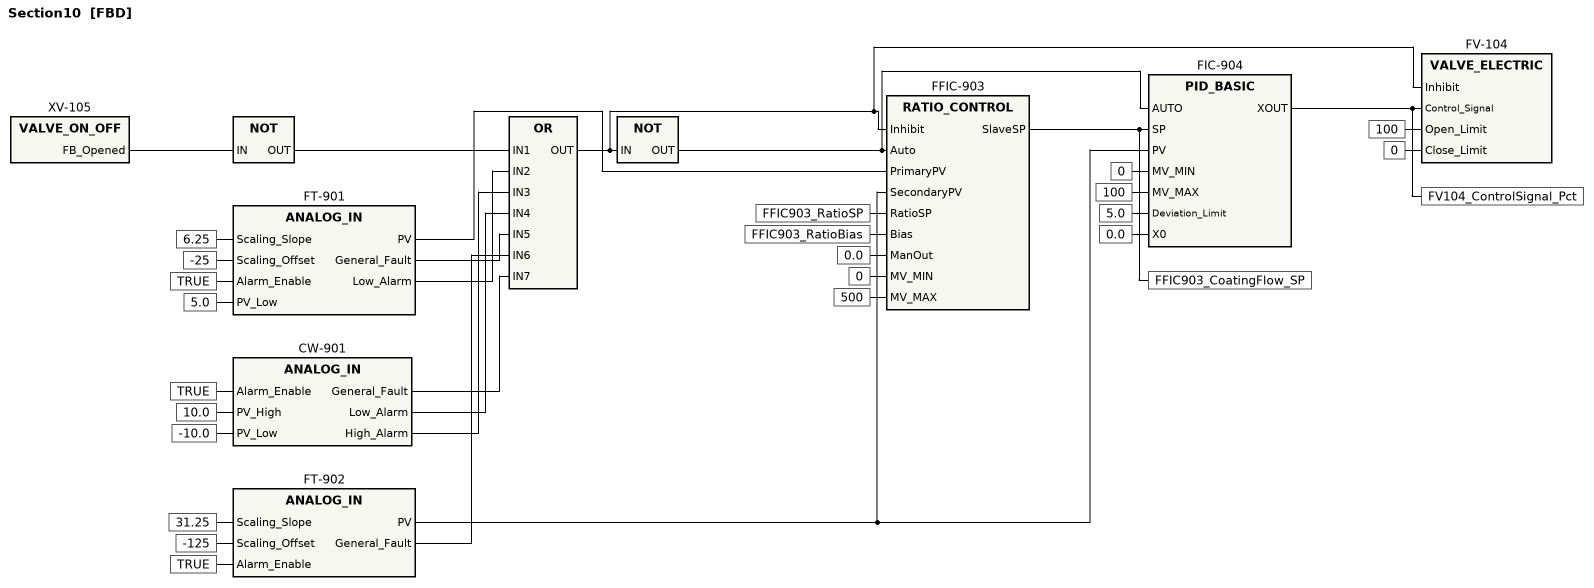
(* FBD diagram, written out as Structured Text *)
XV-105();
FT-901(Scaling_Slope := 6.25, Scaling_Offset := -25, Alarm_Enable := TRUE, PV_Low := 5.0);
CW-901(Alarm_Enable := TRUE, PV_High := 10.0, PV_Low := -10.0);
FT-902(Scaling_Slope := 31.25, Scaling_Offset := -125, Alarm_Enable := TRUE);
_OR497_OUT := NOT XV-105.FB_Opened OR FT-901.Low_Alarm OR CW-901.High_Alarm OR CW-901.Low_Alarm OR FT-901.General_Fault OR FT-902.General_Fault OR CW-901.General_Fault;
_NOT499_OUT := NOT _OR497_OUT;
FFIC-903(Inhibit := _OR497_OUT, Auto := _NOT499_OUT, PrimaryPV := FT-901.PV, SecondaryPV := FT-902.PV, RatioSP := FFIC903_RatioSP, Bias := FFIC903_RatioBias, ManOut := 0.0, MV_MIN := 0, MV_MAX := 500);
FFIC903_CoatingFlow_SP := FFIC-903.SlaveSP;
FIC-904(AUTO := _NOT499_OUT, SP := FFIC-903.SlaveSP, PV := FT-902.PV, MV_MIN := 0, MV_MAX := 100, Deviation_Limit := 5.0, X0 := 0.0);
FV104_ControlSignal_Pct := FIC-904.XOUT;
FV-104(Inhibit := _OR497_OUT, Control_Signal := FIC-904.XOUT, Open_Limit := 100, Close_Limit := 0);
END_PROGRAM

CONFIGURATION Config0
  RESOURCE Res0 ON PLC
    TASK task0(INTERVAL := T#20ms, PRIORITY := 0);
    PROGRAM instance0 WITH task0 : Section2;
    PROGRAM instance_1 WITH task0 : Section3;
    PROGRAM instance_2 WITH task0 : Section4;
    PROGRAM instance_3 WITH task0 : Section5;
    PROGRAM instance_4 WITH task0 : Section6;
    PROGRAM instance_5 WITH task0 : Section7;
    PROGRAM instance_6 WITH task0 : Section8;
    PROGRAM instance_7 WITH task0 : Section9;
    PROGRAM instance_8 WITH task0 : Section10;
  END_RESOURCE
END_CONFIGURATION
